// TIA Portal V18 export
TYPE "UDT_HSsDO"
// stored: IsFailsafeCompliant false
   STRUCT
      xBoilerEnable : Array[1..2] of Bool;
      xBoilerSt1Enable : Array[1..2] of Bool;
      xBoilerSt2Enable : Array[1..2] of Bool;
      xBoilerShuntPumpEnable : Array[1..2] of Bool;
      xBoilerShutOffValveCmd : Array[1..2] of Bool;
   END_STRUCT;
END_TYPE
